{attribute 'linkalways'} 
{attribute 'no_explicit_call' := 'This FB is a CLASS and must be accessed using methods or properties'}
{attribute 'enable_dynamic_creation'}
FUNCTION_BLOCK _ETcVnSvmSgdClassifierType EXTENDS EnumDatatypeBase
VAR
	localData : ETcVnSvmSgdClassifierType;
	activeData : REFERENCE TO ETcVnSvmSgdClassifierType;
	enumBaseDatatype : _DINT(localData);
END_VAR

METHOD PRIVATE AddLocalEnumeration
VAR_INPUT
	Enumeration : T_MAXSTRING;
	Value : ETcVnSvmSgdClassifierType;
END_VAR
AddEnumeration(Enumeration, Value);
END_METHOD

PROPERTY PUBLIC Address : PVOID
GET
Address := ADR(activeData);
END_GET
END_PROPERTY

METHOD PUBLIC ClearReference
VAR_INPUT
END_VAR
activeData REF= localData;
SetBaseDatatypeReference();
END_METHOD

METHOD PUBLIC Clone : I_Datatype
VAR
    pClone : POINTER TO _ETcVnSvmSgdClassifierType;
END_VAR
pClone := __NEW(_ETcVnSvmSgdClassifierType(InitialValue := Value));
Clone := pClone^;
END_METHOD

METHOD FB_init : BOOL
VAR_INPUT
	bInitRetains : BOOL; // if TRUE, the retain variables are initialized (warm start / cold start)
	bInCopyCode : BOOL;  // if TRUE, the instance afterwards gets moved into the copy code (online change)
	InitialValue : ETcVnSvmSgdClassifierType;
END_VAR
localData := InitialValue;
AddBaseDatatype(enumBaseDatatype);
ClearReference();

AddLocalEnumeration('TCVN_SSCT_SGD', ETcVnSvmSgdClassifierType.TCVN_SSCT_SGD);
AddLocalEnumeration('TCVN_SSCT_ASGD', ETcVnSvmSgdClassifierType.TCVN_SSCT_ASGD);
END_METHOD

PROPERTY PUBLIC Identifier : T_MAXSTRING
GET
Identifier := 'ETcVnSvmSgdClassifierType';
END_GET
END_PROPERTY

METHOD IsEnumeratorValueEqual : BOOL
VAR_INPUT
	Enumerator : I_KeyValueForwardEnumerator;
END_VAR
VAR
	storedValue : ETcVnSvmSgdClassifierType;
END_VAR
IF NOT Enumerator.TryGet(storedValue) THEN
	RETURN;
END_IF

IsEnumeratorValueEqual := storedValue = activeData;
END_METHOD

METHOD PUBLIC MakeReferenceTo
VAR_INPUT
	ReferenceTarget : REFERENCE TO ETcVnSvmSgdClassifierType;
END_VAR
activeData REF= ReferenceTarget;
SetBaseDatatypeReference();
END_METHOD

METHOD PROTECTED SetBaseDatatypeReference
VAR_INPUT
END_VAR
enumBaseDatatype.MakeReferenceTo(activeData);
END_METHOD

PROPERTY PUBLIC Size : UDINT
GET
Size := SIZEOF(activeData);
END_GET
END_PROPERTY

METHOD TryMakeReferenceTo : BOOL
VAR_INPUT
	Target : I_Datatype;
END_VAR
VAR
	targetAsEnum : I_EnumDatatype;
	pTargetData : POINTER TO ETcVnSvmSgdClassifierType;
END_VAR
IF NOT Target.TryResolveAsEnumDatatype(targetAsEnum) THEN
	RETURN;
END_IF

IF targetAsEnum.Identifier <> Identifier THEN
	RETURN;
END_IF

pTargetData := Target.Address;
activeData REF= pTargetData^;
SetBaseDatatypeReference();
TryMakeReferenceTo := TRUE;
END_METHOD

PROPERTY PUBLIC Value : ETcVnSvmSgdClassifierType
GET
Value := activeData;
END_GET
SET
activeData := Value;
END_SET
END_PROPERTY

END_FUNCTION_BLOCK

(* stored: Version 1.1.0.1, ProductVersion 3.1.4024.12
   POU _ETcVnSvmSgdClassifierType: Id {5f5abd6b-f2ee-4687-bb63-e0b10bcc2d92}, SpecialFunc None
   Folder Constructor: Id {b3168bea-93f5-4093-9a89-786c6d8a1868}
   Folder Private: Id {6554e9bc-bad6-4fcf-aa9e-245d4e6a0ec6}
   Folder Protected: Id {ee6dbd30-2ad7-4c19-b570-012ac2669256}
   Method AddLocalEnumeration: Id {f1cc9553-e010-4c19-ab30-d283ede93440}
   Property Address: Id {3a87d56c-4fba-4011-84f0-df0814c454ad}
   Get Get: Id {89633f38-f52b-4fb1-89b0-7d78e190e84e}
   Method ClearReference: Id {6e985799-1654-44fc-b273-9d8e54200311}
   Method Clone: Id {8bbad477-b2ae-4e4d-acc5-1e4a81cbb1f4}
   Method FB_init: Id {1f5bfb79-9f5e-4a0b-b42d-b62a52a88efc}
   Property Identifier: Id {d3409e94-567a-4023-9878-e6f0be31163a}
   Get Get: Id {0be05f05-3101-4f80-ba74-a82571095d8e}
   Method IsEnumeratorValueEqual: Id {9f4e84ba-bcd8-4e26-a2ab-0fde63c8a0e9}
   Method MakeReferenceTo: Id {39b69928-b57e-4084-9d0e-1be0a0227c6b}
   Method SetBaseDatatypeReference: Id {9525221f-6270-4e9e-b1f0-e059443f3e39}
   Property Size: Id {759c906c-ef2d-4e29-afcb-b3cfaa433824}
   Get Get: Id {eb8911e8-6900-422b-9a5c-49dd554ee4d3}
   Method TryMakeReferenceTo: Id {b48c1eeb-8041-4bec-a0c5-b89209e9ccaf}
   Property Value: Id {3a0959af-23e6-4fd2-be7f-f29b6315b75e}
   Get Get: Id {f53dcc7e-b755-4c68-92a5-f19757be2456}
   Set Set: Id {41ed1ef1-3b21-4ecd-ac6f-070f50f19197} *)
